INTERFACE I_Domain EXTENDS Debug.I_Debug;

PROPERTY CTable : I_CTable
GET
END_GET
END_PROPERTY

END_INTERFACE

(* stored: Version 1.1.0.1
   Itf I_Domain: Id {c4c62680-655f-41cc-aee4-9ccedbfcc2c8}
   Property CTable: Id {d6197af2-d711-4392-a524-fd934a2b8522}
   Get Get: Id {72b16bc0-4017-476c-ac9f-323e615ee6f9} *)
